PROGRAM MAIN
VAR
	ButtonController : ButtonController;
END_VAR

ButtonController();

END_PROGRAM

(* stored: Version 1.1.0.1, ProductVersion 3.1.4024.12
   POU MAIN: Id {9fb7cb58-d9f1-4206-b911-0a09f555b724}, SpecialFunc None *)
